TYPE "alarmTraceGlobalLevel"
TITLE = Type:Alarm trace global level
VERSION : 1.0
//{"Log": [
//{"version":"v1.0", "date" : "2025-02-01", "author": "cyanezf, "description": "First version"},
//],
//"family":"Alarm",
//"dependencies" : [],
//"description" : "Alarm trace global level"}
//
   STRUCT
      super : UInt;   // 0=No group, 1..N=Super group id
      group : UInt;   // 0=No group, 1..N=Group id
      object : UInt;   // 0=No object; 1..N=Object id
      id : Int;   // 0x0000=No alarm, 0xHHHH=Some alarm
      triggered : Bool;   // 1=Some alarm triggered
      collector : Bool;   // Alarm collector
   END_STRUCT;

END_TYPE

